// TwinCAT 3 PLC project EOL_TESTER
// ProgramVersion: 3.1.4024.0
// libraries:
//   Tc2_Standard, * (Beckhoff Automation GmbH)
//   Tc2_System, * (Beckhoff Automation GmbH)
//   Tc3_Module, * (Beckhoff Automation GmbH)
// project tree:
//   CustomFBs/Actuator/ FB_ActuatorSimple.TcPOU
//   CustomFBs/Actuator/Structure/ ST_ActuatorConfig.TcDUT, ST_ActuatorInputs.TcDUT, ST_ActuatorOutputs.TcDUT, ST_Actuatorstatus.TcDUT
//   CustomFBs/GateBox/ GateBox_FB.TcPOU, ST_MBMStdInput.TcDUT, ST_MGB2IO.TcDUT
//   CustomFBs/MainSequencer/DUT/ ST_MainSequencerStatus.TcDUT
//   CustomFBs/MainSequencer/ MainSequencer.TcPOU
//   CustomFBs/Motor/ FB_Motor.TcPOU, ST_Motor.TcDUT, ST_MotorInputs.TcDUT, ST_MotorStatus.TcDUT
//   CustomFBs/Rockwell_FB/FileLevel/ COP_Dynamic_String_120.TcPOU, COP_Dynamic_String_15.TcPOU, FLL1_String_120.TcPOU, FLL1_String_15.TcPOU
//   CustomFBs/SequenceStep/ FB_SequenceStep.TcPOU, ST_StepBranch_1.TcDUT
//   CustomFBs/SmartLight_BNI007T/ FB_BNI007T.TcPOU, SmartLight.TcDUT, ST_BNI007T.TcDUT
//   / PlcTask.TcTTO
//   POUs/Cell/ Faulthistory_FB.TcPOU, FB_Cell.TcPOU
//   POUs/Cell/ST_Cell/ ST_Cell.TcDUT, ST_CellFaults.TcDUT, ST_CellMode.TcDUT, ST_Error.TcDUT, ST_Estops.TcDUT, ST_Gates.TcDUT, ST_JobSelection.TcDUT, ST_Power.TcDUT, ST_PV_PB.TcDUT, ST_Safety.TcDUT, ST_SmartLight.TcDUT, ST_Status.TcDUT, ST_Utility.TcDUT
//   POUs/Cell/ST_Station/ ST_StaMode.TcDUT, ST_StaRequest.TcDUT, ST_Stastatus.TcDUT, ST_Station.TcDUT
//   POUs/Effenco/ E_CAN_Effenco.TcDUT
//   POUs/ MAIN.TcPOU
//   POUs/SequenceStep_FB/ SequenceStep_FB.TcPOU, ST_StepBranch.TcDUT
//   POUs/Station/TAP/ E_Checkvalvereject.TcDUT, E_PressureStatus.TcDUT, E_PressureTolerance.TcDUT, E_SenorStatus.TcDUT, E_TapAutoSequenceSteps.TcDUT, FB_TAP.TcPOU
//   POUs/Station/TAP/ST_Tap/ ST_TAP_PB.TcDUT (not stored)
// real-time tasks:
//   TASK PlcTask: cycle T#10ms, priority 20, ADS port 350
// I/O:
//   DEVICE Device 1 (EtherCAT), AmsNetId 5.152.37.14.2.1
//     Term 1 (EK1200) [EK1200-5000 EtherCAT Power supply (2A E-Bus)]
//       Term 2 (EL6070) [EL6070 1Ch. Licensing-Terminal]
//       Term 3 (EL6910) [EL6910, TwinSAFE PLC]
//       Term 4 (EL1918) [EL1918, 8Ch. Safety Input 24V, TwinSAFE]
//         modules: Module 1 (FSOE), Module 2 (FSLOGIC)
//       Term 5 (EL1918) [EL1918, 8Ch. Safety Input 24V, TwinSAFE]
//         modules: Module 1 (FSOE), Module 2 (FSLOGIC)
//       Term 6 (EL2904) [EL2904, 4 Ch. Safety Output 24V, 0.5A, TwinSAFE]
//         modules: Module 1 (FSOES), Module 2 (DO)
//       Term 7 (EL2904) [EL2904, 4 Ch. Safety Output 24V, 0.5A, TwinSAFE]
//         modules: Module 1 (FSOES), Module 2 (DO)
//       Term 8 (EL2904) [EL2904, 4 Ch. Safety Output 24V, 0.5A, TwinSAFE]
//         modules: Module 1 (FSOES), Module 2 (DO)
//       Term 9 (EL2904) [EL2904, 4 Ch. Safety Output 24V, 0.5A, TwinSAFE]
//         modules: Module 1 (FSOES), Module 2 (DO)
//       Term 10 (EL9410) [EL9410 E-Bus Power Supplier  (Diagnostics)]
//       Term 11 (EL1008) [EL1008 8Ch. Dig. Input 24V, 3ms]
//       Term 12 (EL2024) [EL2024 4Ch. Dig. Output 24V, 2A]
//       Term 13 (EL6751) [EL6751 CANopen Master]
//       Term 14 (EL6751) [EL6751 CANopen Master]
//       Term 15 (EL9011) [EL9011 End Terminal]
//   DEVICE Device 2 (EL6751), AmsNetId 5.152.37.14.3.1
//   DEVICE Device 3 (EL6751), AmsNetId 5.152.37.14.4.1

CONFIGURATION EOL_TESTER
    RESOURCE PLC ON TwinCAT3
        TASK PlcTask(INTERVAL := T#10ms, PRIORITY := 20);
        PROGRAM MAIN WITH PlcTask : MAIN;
    END_RESOURCE
END_CONFIGURATION

// ---- CustomFBs/Actuator/Structure/ST_ActuatorConfig.TcDUT
TYPE ST_ActuatorConfig :
STRUCT
	AdvancedFeedbackTimeout		: TON;
	RetractedFeedbackTimeout	: TON := (PT := T#500MS);
	AdvancedDwellTime			: TON;
	RetractedDwellTime			: TON;
END_STRUCT
END_TYPE

// ---- CustomFBs/Actuator/Structure/ST_ActuatorInputs.TcDUT
TYPE ST_ActuatorInputs :
STRUCT
	Advanced  AT%I* : BOOL;
	Retracted AT%I* : BOOL;
END_STRUCT
END_TYPE

// ---- CustomFBs/Actuator/Structure/ST_ActuatorOutputs.TcDUT
TYPE ST_ActuatorOutputs :
STRUCT
	Advance  AT%Q* : BOOL;
	Retract  AT%Q* : BOOL;
END_STRUCT
END_TYPE

// ---- CustomFBs/Actuator/Structure/ST_Actuatorstatus.TcDUT
TYPE ST_Actuatorstatus :
STRUCT
	AdvancedFeedback 	: BOOL;
	RetractedFeedback	: BOOL;
	Advancing			: BOOL;
	Retracting			: BOOL;
END_STRUCT
END_TYPE

// ---- CustomFBs/GateBox/ST_MBMStdInput.TcDUT
TYPE ST_MBMStdInput :
STRUCT
    Run_Mode: BIT;  //
END_STRUCT
END_TYPE

// ---- CustomFBs/GateBox/ST_MGB2IO.TcDUT
TYPE ST_MGB2IO :
STRUCT
    
END_STRUCT
END_TYPE

// ---- CustomFBs/MainSequencer/DUT/ST_MainSequencerStatus.TcDUT
TYPE ST_MainSequencerStatus :
STRUCT
	PowerOn 		: BOOL;
	ResetRequired	: BOOL;
	Auto			: BOOL;
	MaintenanceMode	: BOOL;
END_STRUCT
END_TYPE

// ---- CustomFBs/Motor/ST_Motor.TcDUT
TYPE ST_Motor :
STRUCT
    Start_Safeties              : BOOL; //Start Safety
    Start AT%Q*                 : BOOL; //Start
    Running                     : BOOL; //Running
    Stop                        : BOOL; // Motor Stop
    Manual_Start_PB             : BOOL; //Manual Start PV_PB
    Manual_Stop_PB              : BOOL; //Manual Stop PV_PB
    Start_Fault                 : BOOL; //Start_Fault
    OL_Fault                    : BOOL; //Overload_Fault
    Idle_Standby                : BOOL; //Idle_Standby
    Idle_OFF                    : BOOL; //Idle_OFF
    RunOut                      : BOOL; //RunOut
    ONS                         : R_TRIG; //ONS
    
    Motortimedelay              : TON  := (PT := T#2S); //Motor Timer delay
    MotortimeOFFdelay           : TON;
END_STRUCT
END_TYPE

// ---- CustomFBs/Motor/ST_MotorInputs.TcDUT
TYPE ST_MotorInputs :
STRUCT
    Running  AT %I*  : BOOL;  //Assign with Digital Input EL1008
    Overload AT %I*  : BOOL; 
    Enable   AT %I*  : BOOL;
END_STRUCT
END_TYPE

// ---- CustomFBs/Motor/ST_MotorStatus.TcDUT
TYPE ST_MotorStatus :
STRUCT
    Running : BOOL;
END_STRUCT
END_TYPE

// ---- CustomFBs/SequenceStep/ST_StepBranch_1.TcDUT
TYPE ST_StepBranch_1 :
STRUCT    
    NextStep        : DINT;
    Condition       : ARRAY [1..16] OF BOOL;
    ConditionMet    : BOOL;
END_STRUCT
END_TYPE

// ---- CustomFBs/SmartLight_BNI007T/SmartLight.TcDUT
TYPE SmartLight :
STRUCT
    I: SmartLight_BNI007T;
	O: BYTE;
END_STRUCT
END_TYPE

// ---- CustomFBs/SmartLight_BNI007T/ST_BNI007T.TcDUT
TYPE ST_BNI007T :
STRUCT
  	LC_Ok                   : BOOL; 
	RejectPart              : BOOL;   
	InCycle                 : BOOL;	       
	Req_To_Enter_OK         : BOOL;   
	Req_To_Enter_Requested  : BOOL; 
	All_PP                  : BOOL;       
	No_PP                   : BOOL;
	MaintMode               : BOOL;       
	GateLight               : BOOL;
	OperatorLight           : BOOL;
	Station_Enabled         : BOOL;
	Station_Reset           : BOOL;
	Station_At_Load         : BOOL;
	Ready_For_Unload        : BOOL;
	PP_Not_On_Fault         : BOOL;
	PP_Not_Off_Fault        : BOOL;	
	MachineNotRunning       : BOOL;
	GateLocked              : BOOL;
	GateUnlocked            : BOOL;
	AllGatesReset           : BOOL;  
END_STRUCT
END_TYPE

// ---- POUs/Cell/ST_Cell/ST_Cell.TcDUT
TYPE ST_Cell :
STRUCT
	stMode	        : ST_CellMode;
	stUtility	    : ST_Utility;
	stPower	        : ST_Power;
	Status	        : ST_Status;
	PV_PB	        : ST_PV_PB;
	EStop	        : ST_Estops;
	OperatorLight   : ST_SmartLight;
	Job_Selection   : ST_JobSelection;
    Gates           : ST_Gates;
    Faults          : ST_CellFaults;
    Safety          : ST_Safety;
    
END_STRUCT
END_TYPE

// ---- POUs/Cell/ST_Cell/ST_CellFaults.TcDUT
TYPE ST_CellFaults :
STRUCT
FLT_0:BIT; //***WARNING*** DO NOT USE THIS BIT IN LOGIC!!!
FLT_1:BIT; //SAFETY UNLOCKED IN OMRON SAFETY PLC 
FLT_2:BIT; //ETHERNET COMMUNICATION FAULT
FLT_3:BIT; //ETHERNET SWITCHES - FU#  824 TRIPPED
FLT_4:BIT; 
FLT_5:BIT; //GATE 1 - FU# 832 TRIPPED
FLT_6:BIT; //GATE 2 - FU# 834 TRIPPED
FLT_7:BIT; //STATION MASTER BLOCK - FU# 836 TRIPPED
FLT_8:BIT; //CELL MASTER BLOCK - FU# 839 TRIPPED
FLT_9:BIT; //STA10A VALVE BANK POWER - FU# 902 TRIPPED
FLT_10:BIT; //STA10B VALVE BANK POWER - FU# 904 TRIPPED
FLT_11:BIT; //STA20 VALVE BANK POWER - FU# 912 TRIPPED
FLT_12:BIT; //AIR IS OFF - CHECK MAIN AIR DROP
FLT_13:BIT; //GAS IS OFF - CHECK MAIN GAS SWITCH
FLT_14:BIT; //STATION MB - PORT 0 CONNECTION FAULTED
FLT_15:BIT; //STATION MB - PORT 1 CONNECTION FAULTED
FLT_16:BIT; //STATION MB - PORT 2 CONNECTION FAULTED
FLT_17:BIT; //STATION MB - PORT 3 CONNECTION FAULTED
FLT_18:BIT; //STATION MB - PORT 4 CONNECTION FAULTED
FLT_19:BIT; //STATION MB - PORT 5 CONNECTION FAULTED
FLT_20:BIT; //STATION MB - PORT 6 CONNECTION FAULTED
FLT_21:BIT; //STATION MB - PORT 7 CONNECTION FAULTED
FLT_22:BIT; //CELL MB - PORT 0 CONNECTION FAULTED
FLT_23:BIT; //CELL MB - PORT 1 CONNECTION FAULTED
FLT_24:BIT; //CELL MB - PORT 2 CONNECTION FAULTED
FLT_25:BIT; //CELL MB - PORT 3 CONNECTION FAULTED
FLT_26:BIT; //CELL MB - PORT 4 CONNECTION FAULTED
FLT_27:BIT; //CELL MB - PORT 5 CONNECTION FAULTED
FLT_28:BIT; //CELL MB - PORT 6 CONNECTION FAULTED
FLT_29:BIT; //CELL MB - PORT 7 CONNECTION FAULTED
FLT_30:BIT; 
FLT_31:BIT; 
FLT_32:BIT; 
FLT_33:BIT; 
FLT_34:BIT; 
FLT_35:BIT; 
FLT_36:BIT; 
FLT_37:BIT; 
FLT_38:BIT;
FLT_39:BIT;
FLT_40:BIT; //HMI ESTOP WAS DEPRESSED
FLT_41:BIT; //HMI ESTOP INPUTS INCONSISTENT
FLT_42:BIT; //MHR1 LOCAL ESTOP WAS DEPRESSED
FLT_43:BIT; //MHR1 LOCAL ESTOP INPUTS INCONSISTENT
FLT_44:BIT;
FLT_45:BIT; //OPERATOR ESTOP WAS DEPRESSED
FLT_46:BIT; //OPERATOR ESTOP INPUTS INCONSISTENT
FLT_47:BIT; //OPERATOR 2 RH ESTOP WAS DEPRESSED
FLT_48:BIT; //OPERATOR 2 RH ESTOP INPUTS INCONSISTENT
FLT_49:BIT;
FLT_50:BIT; //GATE 1 ESTOP WAS DEPRESSED
FLT_51:BIT; //GATE 2 ESTOP WAS DEPRESSED
FLT_52:BIT; 
FLT_53:BIT; 
FLT_54:BIT; 
FLT_55:BIT; 
FLT_56:BIT; 
FLT_57:BIT; 
FLT_58:BIT; 
FLT_59:BIT;
FLT_60:BIT; 
FLT_61:BIT; 
FLT_62:BIT; 
FLT_63:BIT; 
FLT_64:BIT;
FLT_65:BIT; 
FLT_66:BIT; 
FLT_67:BIT; 
FLT_68:BIT; 
FLT_69:BIT; //SAFETY GATE 1 NOT IN RUN MODE
FLT_70:BIT; //SAFETY GATE 1 UNLOCKED
FLT_71:BIT; 
FLT_72:BIT; //SAFETY GATE 1 DOOR OPENED
FLT_73:BIT; 
FLT_74:BIT; //SAFETY GATE 2 NOT IN RUN MODE
FLT_75:BIT; //SAFETY GATE 2 UNLOCKED
FLT_76:BIT; 
FLT_77:BIT; //SAFETY GATE 2 DOOR OPENED
FLT_78:BIT; 
FLT_79:BIT; 
FLT_80:BIT; //LIGHT CURTAIN INPUTS INCONSISTENT
FLT_81:BIT; //LIGHT CURTAIN EDM ERROR
FLT_82:BIT; //LIGHT CURTAIN NOT OK
FLT_83:BIT; //LIGHT CURTAIN IN ERROR STATE
FLT_84:BIT; 
FLT_85:BIT; 
FLT_86:BIT; 
FLT_87:BIT; 
FLT_88:BIT; 
FLT_89:BIT; //OMRON SAFETY PROCESSOR NOT MATCHING 
FLT_90:BIT; //HMI POINT IO - COMMUNICATION FAULT
FLT_91:BIT; //OMRON SAFETY PLC - COMMUNICATION FAULT
FLT_92:BIT; //STATION MASTER IO BLOCK - COMMUNICATION FAULT
FLT_93:BIT; //CELL MASTER IO BLOCK - COMMUNICATION FAULT
FLT_94:BIT; //SAFETY GATE 1 - COMMUNICATION FAULT
FLT_95:BIT; //SAFETY GATE 2 - COMMUNICATION FAULT
END_STRUCT
END_TYPE

// ---- POUs/Cell/ST_Cell/ST_CellMode.TcDUT
TYPE ST_CellMode :
STRUCT
	Manual 				: BOOL;         //IN MANUAL MODE
	Auto				: BOOL;         //IN AUTO MODE
	Supervisor_Mode 	: BOOL;         //IN SUPERVISOR MODE
    AutoSelect_Toggle   : um_Toggle;    //Auto Select Toggle
    Autoinitiate         :BOOL;          //Cell Auto Initiate
	In_DryCycle_Select 	: BOOL;         //IN DRY CYCLE MODE
	DryCycle_Runout		: BOOL;         //DRY CYCLE RUN OUT
	DryCycle_ONS		: R_TRIG;       //DRY CYCLE (ONE SHOT)
	In_Continuous_Run	: BOOL;         //IN CONTINUOUS RUN
	Continuos_Run_ONS	: R_TRIG;       //CONTINUOUS RUN (ONE SHOT)
END_STRUCT
END_TYPE

// ---- POUs/Cell/ST_Cell/ST_Error.TcDUT
TYPE ST_Error :
STRUCT
    Active      : BOOL;
    Message     : STRING;
    Priority    : UDINT;
END_STRUCT
END_TYPE

// ---- POUs/Cell/ST_Cell/ST_Estops.TcDUT
TYPE ST_Estops :
STRUCT
Gate1:BIT; 
Gate2:BIT; 
Gate3:BIT; 
Gate4:BIT; 
Gate5:BIT; 
Gate6:BIT; 
Oper1:BIT; 
Oper2:BIT; 
Oper3:BIT; 
Oper4:BIT; 
Oper5:BIT; 
Oper6:BIT; 
Main_Panel:BIT; 
HMI_Panel:BIT; 
Any_EStop_PB_Pressed: BIT;
Local_EStop_1_PB_Pressed: BIT;
END_STRUCT
END_TYPE

// ---- POUs/Cell/ST_Cell/ST_Gates.TcDUT
TYPE ST_Gates :
STRUCT
    //Gate Box
    Request_To_Enter             : BOOL;                  //Request to Enter
    Reset                        : ARRAY [1..5] OF BOOL;  //Reset Door
    Resume_ONS                   : R_TRIG;                //Resume(One Shot)
    OK_To_Enter                  : BOOL;                  //Ok to Enter (Station)
    EntryGranted                 : BOOL;                  //Granted (Unlock Doors)
    EStop_Mem                    : BOOL;
    Closed                       : BOOL;
    Teach_Mode_OK                : BOOL; 
    
    //Gate SAFTY OUTPUT
    DoorUnlockRequest            : ARRAY [1..5] OF BOOL; //Door Unlock Request
    DoorOktoUnlock               : ARRAY [1..5] OF BOOL; //Door Ok to Unlcok
    ReqtoEnterInput_LT  AT%Q*    : ARRAY [1..5] OF BOOL; //WHITE Light  Requst to Enter (Input)     
    FaultResetInput_LT  AT%Q*    : ARRAY [1..5] OF BOOL; //RED Light    Door Fault Reset
    PowerOn_LT          AT%Q*    : ARRAY [1..5] OF BOOL; //GREEN Light  Door Power ON/Cycle start Input
    
    //Gate SAFETY INPUT
    Run_Mode                                    : BIT;//SI_RM
	Connection_Fauled                           : BIT;//SI_CF
	Diagnostic_Active                           : BIT;//SI_DA
	FailSafe_Input_EStop_OK                     : BIT;//SI_FIES
	FailSafe_Input_DoorPosition                 : BIT;//SI_FI_D
	FailSafe_Input_BoltPosition                 : BIT;//SI_FI_B
	FailSafe_Input_GuardLocking                 : BIT;//SI_FI_L (GATE LOCKED)
	FailSafe_Input_DoorAndBolt_Position         : BIT;//SI_FI_SK
	FailSafe_Input_DoorBoltAndGuardLocking      : BIT;//SI_FI_UK
	Maintenance_Mode                            : BIT;//SI_S94
    DoorReqtoEnterInput AT%I*                   : ARRAY [1..5] OF BOOL; //SI_S2//WHITE PB  Requst to Enter (Input)     
    DoorFaultResetInput AT%I*                   : ARRAY [1..5] OF BOOL; //SI_S3//RED PB    Door Fault Reset
    DoorPowerOn         AT%I*                   : ARRAY [1..5] OF BOOL; //SI_S4//GREEN PB  Door Power ON/Cycle start Input
	Diagnostics_Plausibility_Fault              : BIT;//SI_D_PF
	Diagnostics_Emergency_Stop                  : BIT;//SI_D_ES
	Diagnostics_GuardLocking                    : BIT;//SI_D_OL
	Diagnostics_Lifetime                        : BIT;//SI_D_LT

    
END_STRUCT                          
END_TYPE

// ---- POUs/Cell/ST_Cell/ST_JobSelection.TcDUT
TYPE ST_JobSelection :
STRUCT
Auto_Job_Mode			: BOOL;
Part_Sel_Chng_OK		: BOOL;
HMI_Selected_Job		: DINT;
Job_Number_Selected		: DINT;
Job_Number_Selected_Last: DINT;
Job_Change_Started		: BOOL;
Job_Change_Delay		: TON;	
END_STRUCT
END_TYPE

// ---- POUs/Cell/ST_Cell/ST_Power.TcDUT
TYPE ST_Power :
STRUCT
Gen_Safety	:BOOL;		//General_Safety_OK(COntrol POwer)(Gate Closed)(Air OK)
PowerOn		:BOOL; 		//CONTROL POWER ON
EStops		:ST_Estops;	//NO E-STOPS BUTTONS PRESSED
GatesClosed	:BOOL; 		//CELL SAFETY GATES CLOSED & RESET
END_STRUCT
END_TYPE

// ---- POUs/Cell/ST_Cell/ST_PV_PB.TcDUT
TYPE ST_PV_PB :
STRUCT
	FaultReset_PB 		:BOOL;  //FAULT_RESET PV_PB
	AutoManual_SS 		:BOOL; 	//AUTO/MANUAL SELECTOR SWITCH PV PB
	AutoSelector_PB 	:BOOL; 	//AUTO_SELECTOR SWITCH PV PB
	ManualSelector_PB 	:BOOL; 	//MANUAL_SELECTOR SWITCH PV PB
	AutoMode_PB		:BOOL; 	//AUTO MODE PV PB
	Dry_Cycle_Mode		:BOOL;	//DRY_CYCLE_MODE PV PB
	ContinousRun_Mode	:BOOL;	//CONTINUOUS RUN MODE PV PB
	FaultHistory_Reset	:BOOL;	//FAULT HISTOTY RESET PV PB
END_STRUCT
END_TYPE

// ---- POUs/Cell/ST_Cell/ST_Safety.TcDUT
TYPE ST_Safety :
STRUCT
    MCPEstopOk AT%I*  : BOOL;
    SafetyOk AT%I*    : BOOL;
    
END_STRUCT
END_TYPE

// ---- POUs/Cell/ST_Cell/ST_SmartLight.TcDUT
TYPE ST_SmartLight :
STRUCT
	Green			: BOOL;  
	Process_Fault	: BOOL;
	InCycle			: BOOL;
	Blue			: BOOL;
	Orange			: BOOL;
	White			: BOOL;
    Flash			: BOOL;	
END_STRUCT
END_TYPE

// ---- POUs/Cell/ST_Cell/ST_Status.TcDUT
TYPE ST_Status :
STRUCT
AllComms_OK		:BOOL; //ALL COMMUNICATION MODULES OK
ENetComms_OK    :BOOL; //All EtherCAT Comms Ok
Faulted			:BOOL; //Fault(s) Present
Fault_Reset		:BOOL; //Fault Reset
All_Faults		:BOOL; //ANY STATION FAULTED
All_in_Auto		:BOOL; //ALL_STATIONS IN AUTO MODE
All_in_Manuals	:BOOL; //ALL_SATIONS_IN MANUAL MODE
StationsHeld	:BOOL; //Station is Hold in between Test
Held			:BOOL; //CELL HOLD BUTTON PRESSED
Message			:BOOL; //Message(s) Present
ProcessOn		:BOOL; //DUT (Device Under Test) is ON
ProcessOff		:BOOL; //DUT (Device Under Test) is OFF
OKToEnterGates	:BOOL; //Safe
END_STRUCT
END_TYPE

// ---- POUs/Cell/ST_Cell/ST_Utility.TcDUT
TYPE ST_Utility :
STRUCT
MainAirOn	     :BOOL;        //MAIN AIR PRESSURE OK
MainAirPSI AT%I* :REAL;        //MAIN AIR DATA FROM BALLUFF PRESSURE SENSOR
END_STRUCT
END_TYPE

// ---- POUs/Cell/ST_Station/ST_StaMode.TcDUT
TYPE ST_StaMode :
STRUCT
    ManualReady             : BIT; //READY FOR MANUAL
    Manual                  : BIT;//IN MANUAL MODE
    AutoReady               : BIT; //READY FOR AUTO
    Auto                    : BIT; //IN AUTO MODE
    DryCycleReady           : BIT; // READY FOR DRYCYCLE
    DryCycle                : BIT; //IN DRY CYCLE MODE (RUN EMPTY)
    PartTest                : BIT; //WHITE RABBIT TEST MODE
    AutoWarning             : TON; // AUTO WARNING TIMER
    Job_Select_PB           : BIT;// JOB SELECT PUSHBUTTON
END_STRUCT
END_TYPE

// ---- POUs/Cell/ST_Station/ST_StaRequest.TcDUT
TYPE ST_StaRequest :
STRUCT
    AutoInitiate        : BIT; // 
    AutoConfirm         : BIT; // 
    FaultReset          : BIT; // 
    Hold                : BIT; // 
    LampTest            : BIT; // 
    PauseMSG            : BIT; // 
    DryCycle            : BIT; // 
    AllProcessOn        : BIT; // 
    AllProcessOff       : BIT; // 
    ProdCountReset      : BIT; //   
END_STRUCT
END_TYPE

// ---- POUs/Cell/ST_Station/ST_Stastatus.TcDUT
TYPE ST_Stastatus :
STRUCT
    AirOff                  : BIT; // 
    AirOn                   : BIT; // 
    AllParts                : BIT; // STATION HAS ALL PARTS PRESENT 
    AllProcessesComplete    : BIT; // ALL PROCESSES COMPLETE
    All_Tools_In_Known_Pos  : BIT; //
    All_Faults              : BIT;// 
    Auto                    : BIT; // STATION IN AUTO
    ClearForTransfer        : BIT; // 
    CommOK                  : BIT; // STATION COMMUNICATIONS ARE OK
    DryCycle                : BIT; // STATION IN DRY CYCLE
    Faulted                 : BIT; // STATION FAULTED
    GasFlowOff              : BIT; // 
    GasFlowOn               : BIT; // 
    Held                    : BIT; // STATION HELD
    HoldActive              : BIT; // STATION HOLD IS ACTIVE
    Home                    : BIT; // TOOL AT HOME POSITION
    InCycle                 : BIT; // STATION IN CYCLE
    Load1                   : BIT; // TOOL AT LOAD POSITION 1
    Load2                   : BIT; // TOOL AT LOAD POSITION 2
    Manual                  : BIT; // STATION IN MANUAL
    Message                 : BIT; // Message(s) Present
    NoParts                 : BIT; // STATION HAS NO PARTS PRESENT
    NoProcComp              : BIT; // NO PROCESS COMPLETE
    NotClear                : BIT; // 
    OK_To_Enter             : BIT; // Clear To Enter if Gate Request Has Been Made
    PartPres                : BIT; // 
    Proc1Comp               : BIT; // 1st PROCESS COMPLETE
    Proc2Comp               : BIT; // 2nd PROCESS COMPLETE
    Proc3Comp               : BIT; // 3rd PROCESS COMPLETE
    Proc4Comp               : BIT; // 4th PROCESS COMPLETE
    Proc5Comp               : BIT; // 5th PROCESS COMPLETE
    Proc6Comp               : BIT; // 6th PROCESS COMPLETE
    Proc7Comp               : BIT; // 7th PROCESS COMPLETE
    Proc8Comp               : BIT; // 8th PROCESS COMPLETE
    ProcEnbld               : BIT; // 
    ProcNotEnbld            : BIT; // 
    Sla01_ID                : BYTE; // ID PRESENT ON SLAVE#1
    Sla02_ID                : BYTE; // ID PRESENT ON SLAVE#2
    SteppersReset           : BIT; // 
    Tool_Monitor            : DINT;
    Unload1                 : BIT; // TOOL AT UNLOAD POSITION 1
    UnLoad2                 : BIT; // TOOL AT UNLOAD POSITION 2
    WaterFlowOff            : BIT; // 
    WaterFlowOn             : BIT; // 
    Work1                   : BIT; // TOOL AT WORK POSITION 1
    Work2                   : BIT; // TOOL AT WORK POSITION 2
    Work3                   : BIT; // TOOL AT WORK POSITION 3
END_STRUCT
END_TYPE

// ---- POUs/Cell/ST_Station/ST_Station.TcDUT
TYPE ST_Station :
STRUCT
    Mode        : ST_StaMode;                   // Station Mode
    Status      : ST_Stastatus;                // Station Status 
    Req         : ST_StaRequest;               // 
END_STRUCT
END_TYPE

// ---- POUs/Effenco/E_CAN_Effenco.TcDUT
{attribute 'qualified_only'}
{attribute 'strict'}
TYPE E_CAN_Effenco :
(
	enum_member := 0
);
END_TYPE

// ---- POUs/SequenceStep_FB/ST_StepBranch.TcDUT
TYPE ST_StepBranch :
STRUCT    
    NextStep        : DINT;
    Condition       : ARRAY [1..16] OF BOOL;
    ConditionMet    : BOOL;
END_STRUCT
END_TYPE

// ---- POUs/Station/TAP/E_Checkvalvereject.TcDUT
{attribute 'qualified_only'}
{attribute 'strict'}
TYPE E_Checkvalvereject :
(
	enum_member         := 0,
    CheckvalveOk        := 10,
    Checkvalvefailure   := 20
);
END_TYPE

// ---- POUs/Station/TAP/E_PressureStatus.TcDUT
{attribute 'qualified_only'}
{attribute 'to_string'}
TYPE E_PressureStatus : 
(
    FillingupTestFail    := 10,
    FillingupTestPass    := 20,
    PressuretestOk       := 30,
    Pressuretestfail     := 40,
    InletLeakDetect      := 50,
    OilLeakDetect        := 60
    	
);
END_TYPE

// ---- POUs/Station/TAP/E_PressureTolerance.TcDUT
{attribute 'qualified_only'}
{attribute 'strict'}
TYPE E_PressureTolerance :
(
	enum_member := 0
);
END_TYPE

// ---- POUs/Station/TAP/E_SenorStatus.TcDUT
{attribute 'qualified_only'}
{attribute 'strict'}
TYPE E_SenorStatus :
(
	enum_member         := 0,
    P1UUTSensorOK       := 10,
    P1UUTSensorFail     := 20,
    P2UUTSensorOK       := 30,
    P2UUTSensorFail     := 40,
    Filterisdetected    := 50,
    Filterismissing     := 60
    
    
);
END_TYPE

// ---- POUs/Station/TAP/E_TapAutoSequenceSteps.TcDUT
{attribute 'qualified_only'}
{attribute 'strict'}
TYPE E_TapAutoSequenceSteps :
(
	STARTING_CONDITIONS		    := 10,
    START_FILLING_PHASE 	    := 20,
	TE_RUN_MOTOR			    := 30,
//	TE_MOTOR_START_DELAY	    := 40,
	START_UUT_MOTOR			    := 50,
	UUT_MOTOR_DELAY			    := 60,
	INITIAL_PRESSURE_TEST	    := 70,
    TE_STOP_MOTOR               := 80,
    STOP_UUT_MOTOR              := 90,
    END_FILLING_PHASE           := 100,
    START_STATIC_PRESSURE_TEST  := 110,
    OUTLET_PRESSURE_TEST        := 120,
    OIL_LEAK_TEST               := 130,
    END_STAITC_PRESSURE_TEST    := 140,
    START_FUNCTIONAL_TEST       := 150,
    UUT_SENSOR_CHECK            := 160,
    END_FUNCTIONAL_TEST         := 170,
    START_TAP_CHECKVALVE_TEST   := 180,
    CHECK_VALVE_TEST            := 190,
    END_TAP_CHECKVALVE_TEST     := 200,
    START_DRAINING_TEST         := 210, 
    STOP_DRAINING_TEST          := 220,    
    COMPLETE                := 1000
	
);
END_TYPE

// ---- POUs/MAIN.TcPOU
PROGRAM MAIN
VAR
END_VAR

END_PROGRAM

// ---- CustomFBs/Actuator/FB_ActuatorSimple.TcPOU
FUNCTION_BLOCK FB_ActuatorSimple
VAR_INPUT
    stCell      : ST_Cell;
    stStation   : ST_Station;
END_VAR
VAR
	stStatus			: ST_Actuatorstatus;
	stConfiguration 	: ST_ActuatorConfig;
	stInputs			: ST_ActuatorInputs;
	stOutputs			: ST_ActuatorOutputs;
END_VAR

//_M_EvaluateInputs();
_M_Status();

METHOD PRIVATE _M_EvaluateInputs
VAR_INPUT
END_VAR
END_METHOD

METHOD PUBLIC _M_Status : BOOL
VAR_INPUT
END_VAR
// Reset Status
//Status.AdvancedFeedback := FALSE;
//Status.Advancing := FALSE;
//Status.RetractedFeedback := FALSE;
//Status.Retracting := FALSE;

// Set According To Raw Value
IF stInputs.Advanced AND NOT stInputs.Retracted THEN
    stStatus.AdvancedFeedback := TRUE;
    stConfiguration.AdvancedFeedbackTimeout(IN:=FALSE);
    IF stOutputs.Advance THEN
        stOutputs.Advance := FALSE;
    END_IF
ELSE
    IF stOutputs.Advance THEN
        stStatus.Advancing := TRUE;
    END_IF
END_IF	

IF stInputs.Retracted AND stInputs.Advanced THEN 	
    stStatus.RetractedFeedback := TRUE;
    IF stOutputs.Retract THEN
        stOutputs.Retract := FALSE;
    END_IF
ELSE
    IF stOutputs.Retract THEN
        stStatus.Retracting := TRUE;
    END_IF
END_IF

IF stInputs.Advanced AND stInputs.Retracted THEN
    //error handling
END_IF
END_METHOD

METHOD PUBLIC M_Advance
//At Advance Position

IF stStatus.RetractedFeedback AND NOT stStatus.AdvancedFeedback THEN      
      stOutputs.Retract := FALSE;
      stOutputs.Advance := TRUE;
      stConfiguration.AdvancedFeedbackTimeout(IN:=TRUE);
END_IF      
IF NOT stStatus.AdvancedFeedback AND stConfiguration.AdvancedFeedbackTimeout.Q THEN
    //time out happened - indicate fault
    //reset output for advance and retract
    //monitor safety
END_IF
END_METHOD

METHOD PUBLIC M_Retract
VAR_INPUT
END_VAR
//At Retract Position
END_METHOD

PROPERTY PUBLIC P_Config : REFERENCE TO ST_ActuatorConfig
GET // PUBLIC
P_Config REF= stConfiguration;
END_GET
END_PROPERTY

PROPERTY PUBLIC P_Status : REFERENCE TO ST_Actuatorstatus
GET
P_Status REF= stStatus;
END_GET
END_PROPERTY

END_FUNCTION_BLOCK

// ---- CustomFBs/GateBox/GateBox_FB.TcPOU
FUNCTION_BLOCK GateBox_FB
VAR 
    Gate1   : ST_Gates;
    Gate2   : ST_Gates;
END_VAR

//GateBox-1 Lock Solenoid
IF GVL.stCell.Gates.DoorReqtoEnterInput[1] AND GVL.stCell.Gates.Request_To_Enter THEN
    GVL.stCell.Gates.DoorUnlockRequest[1] := TRUE;
ELSIF GVL.stCell.Gates.DoorPowerOn[1] AND  GVL.zz_Deep.0 AND GVL.zz_Deep.0 THEN
    GVL.stCell.Gates.DoorUnlockRequest[1] := FALSE;
END_IF

GVL.stCell.Gates.DoorOktoUnlock[1] := (GVL.stCell.Gates.EntryGranted OR 
                                          GVL.stCell.Gates.DoorOktoUnlock[1] OR 
                                          GVL.zz_Deep.0)  AND 
                                          GVL.stCell.Gates.DoorUnlockRequest[1];
                                         
//GateBox-1 - Smart light Mapping
//White Light
GVL.stCell.Gates.ReqtoEnterInput_LT[1] :=  GVL.stCell.Gates.DoorUnlockRequest[1] AND 
                                            GVL.stCell.Gates.Request_To_Enter AND 
                                            GVL.stCell.Gates.OK_To_Enter AND 
                                            GVL.stCell.Gates.EntryGranted AND 
                                            (NOT Gate1.Maintenance_Mode OR (Gate1.Maintenance_Mode AND Gate1.Teach_Mode_OK));  

//Green Liight
GVL.stCell.Gates.FaultResetInput_LT[1] :=  (Gate1.Reset OR (Gate1.closed AND NOT Gate1.Reset AND Gate1.Maintenance_Mode) AND 
                                            (NOT Gate1.Maintenance_Mode OR (Gate1.Maintenance_Mode AND Gate1.Teach_Mode_OK)))  OR
                                            (Gate1.Maintenance_Mode AND NOT Gate1.Teach_Mode_OK);
                                            
                                            
//Red Light
GVL.stCell.Gates.FaultResetInput_LT[1] :=  (GVL.stCell.Status.All_Faults AND 
                                            ( NOT Gate1.Maintenance_Mode OR (Gate1.Maintenance_Mode AND Gate1.Teach_Mode_OK))) OR
                                            Gate1.DoorFaultResetInput   OR
                                            (Gate1.Maintenance_Mode AND NOT Gate1.Teach_Mode_OK);
                                            

                                            
                                            
                                            
                                            
//GateBox-2 Lock Solenoid
IF GVL.stCell.Gates.DoorReqtoEnterInput[2] AND GVL.stCell.Gates.Request_To_Enter THEN
    GVL.stCell.Gates.DoorUnlockRequest[2] := TRUE;
ELSIF GVL.stCell.Gates.DoorPowerOn[1] AND  GVL.zz_Deep.0 AND GVL.zz_Deep.0 THEN
    GVL.stCell.Gates.DoorUnlockRequest[2] := FALSE;
END_IF

GVL.stCell.Gates.DoorOktoUnlock[2] := (GVL.stCell.Gates.EntryGranted OR 
                                          GVL.stCell.Gates.DoorOktoUnlock[2] OR 
                                          GVL.zz_Deep.0)  AND 
                                          GVL.stCell.Gates.DoorUnlockRequest[2];

//GateBox-2 - Smart light Mapping
//White Light
GVL.stCell.Gates.ReqtoEnterInput_LT[2] :=  GVL.stCell.Gates.DoorUnlockRequest[2] AND 
                                            GVL.stCell.Gates.Request_To_Enter AND 
                                            GVL.stCell.Gates.OK_To_Enter AND 
                                            GVL.stCell.Gates.EntryGranted AND 
                                            (NOT Gate2.Maintenance_Mode OR (Gate2.Maintenance_Mode AND Gate2.Teach_Mode_OK));  

//Green Liight
GVL.stCell.Gates.FaultResetInput_LT[2] :=  (Gate2.Reset OR (Gate2.closed AND NOT Gate2.Reset AND Gate2.Maintenance_Mode) AND 
                                            (NOT Gate2.Maintenance_Mode OR (Gate2.Maintenance_Mode AND Gate2.Teach_Mode_OK)))  OR
                                            (Gate2.Maintenance_Mode AND NOT Gate2.Teach_Mode_OK);
                                            
                                            
//Red Light
GVL.stCell.Gates.FaultResetInput_LT[2] :=  (GVL.stCell.Status.All_Faults AND 
                                            ( NOT Gate2.Maintenance_Mode OR (Gate2.Maintenance_Mode AND Gate2.Teach_Mode_OK))) OR
                                            Gate2.DoorFaultResetInput   OR
                                            (Gate2.Maintenance_Mode AND NOT Gate2.Teach_Mode_OK)

END_FUNCTION_BLOCK

// ---- CustomFBs/MainSequencer/MainSequencer.TcPOU
FUNCTION_BLOCK MainSequencer
VAR_INPUT
	Status	: REFERENCE TO ST_MainSequencerStatus;
END_VAR
VAR
	fbTest1Sequencer	: Test1Sequencer;	
	oPowerPackChargeRequest	 AT%Q* : BOOL;
END_VAR

_M_Test1();
//_M_AutoSequence();

METHOD PRIVATE _M_AutoSequence
VAR_INPUT
END_VAR
fbTest1Sequencer.M_AutoSequence(AutoSteps := E_Test1AutoSteps.PRESSURIZEHYDRAULICMOTOR);
END_METHOD

METHOD PRIVATE _M_Test1
VAR_INPUT
END_VAR
fbTest1Sequencer();
END_METHOD

END_FUNCTION_BLOCK

// ---- CustomFBs/Motor/FB_Motor.TcPOU
FUNCTION_BLOCK FB_Motor
VAR_INPUT
   SafetyOk               : BOOL;
END_VAR
VAR 
    stMotor               : ST_Motor;
    stMotorInputs         : ST_MotorInputs;
    Error                 : ST_Error (Priority := 999);
    Status                : ST_MotorStatus;
END_VAR


(* Monitoring all Digital Inputs during Process *)
M_Monitor();

(* HPU - Faults *)
M_Fault();

METHOD PRIVATE M_Fault : BOOL
VAR_INST
    (*Fault Timers*)
    System_Faults       : ARRAY [0..10] OF BOOL;
	Fault_Tmrs          : ARRAY [0..10] OF TON;
END_VAR
VAR
    Error : ST_Error;
END_VAR
 Error.Active := stMotorInputs.Overload;
 Error.Message := 'Motor Overload Tripped';
 M_RaiseError(InputError := Error);



   (*Fault1 - HPU Enable input not coming on: check relay in MCP Panel*)
		Fault_Tmrs[1].PT:= T#2.5S;
		Fault_Tmrs[1]();
		Fault_Tmrs[1].IN:=  GVL.zz_Deep.0 AND //need to add safety EDM condition 
							  stMotorInputs.Enable ;
        System_Faults[1]:= Fault_Tmrs[1].Q;
        
    (*Fault2 - HPU Running Input is not coming ON *)
		Fault_Tmrs[2].PT:= T#2.5S;
		Fault_Tmrs[2]();
		Fault_Tmrs[2].IN:= stMotor.Start AND
                              stMotorInputs.Running; 
        System_Faults[2]:= Fault_Tmrs[2].Q;    
        
    (*Fault3 - HPU Motor OverLoad Trip: CheckUnit *)
		Fault_Tmrs[3].PT:= T#0.5S;
		Fault_Tmrs[3]();
		Fault_Tmrs[3].IN:= stMotorInputs.Overload;  
        System_Faults[3]:= Fault_Tmrs[].Q;  
        
   (*Fault4 - Low Critical Oil: Motor can not run until Tank is Filled *)
		Fault_Tmrs[].PT:= T#0.5S;
		Fault_Tmrs[]();
		Fault_Tmrs[].IN:= ;  
        System_Faults[]:= Fault_Tmrs[].Q;
        
   (*Fault5 - Oil Temperature Critical: Motor Can not run until Oil Cools Down *)
		Fault_Tmrs[].PT:= T#0.5S;
		Fault_Tmrs[]();
		Fault_Tmrs[].IN:=   
        System_Faults[]:= Fault_Tmrs[].Q;
        
    (*Fault6 - HPU High Pressure Bypass Valve Faulted - not going to Low Pressure: Major Fault *)
		Fault_Tmrs[].PT:= T#12.5S;
		Fault_Tmrs[]();
		Fault_Tmrs[].IN:=  
        System_Faults[]:= Fault_Tmrs[].Q;
END_METHOD

METHOD PRIVATE M_Monitor : BOOL
VAR   
END_VAR

//Do we still need to monitor even if we are monitoring in faults

//IF stMotor.Start  THEN    //Should I add more condition from safety related to CH-1 and CH-2
//     stMotorInputs.Running AND stMotorInputs.Enable AND NOT stMotorInputs.Overoload
  
//END_IF


//Do we need to monitro safety input here as well?
END_METHOD

METHOD PRIVATE M_RaiseError
VAR_INPUT
    InputError : ST_Error;
END_VAR
IF InputError.Priority < Error.Priority THEN
    Error := InputError;
END_IF
END_METHOD

METHOD PUBLIC M_ResetFault
VAR
    NullError : ST_Error;
END_VAR
Error := NullError;
END_METHOD

METHOD M_Start : BOOL
VAR

    SafetyNOKError : ST_Error (Message := 'Motor Not Started Fault Due To Safety NOK', Priority := 1); 
    
END_VAR
 //Verify Motor Safety
 
(*IF  SafetyOk  AND                                 //tHIS CONDITION WILL MONITOR BEFORE RUN MOTOR PROGRAM    
         NOT stMotorInputs.Overload AND            //OL Relay Tripped Input
         NOT M_Fault(); THEN                    //Need to verify this logic
    stMotor.Start_Safeties := TRUE;
ELSE
    stMotor.Start_Safeties := FALSE;
END_IF*)          
         
IF (stStation.Mode.Auto OR    
         (stStation.Mode.Manual AND 
            stMotor.Manual_Start_PB)) AND 
                stMotor.Start_Safeties THEN
    stMotor.Start := TRUE;
    stmotor.Motortimedelay (IN := TRUE);   
ELSE
     

IF SafetyOk THEN
    stMotor.Start := TRUE;
ELSE    
    stMotor.Start := FALSE;
    SafetyNOKError.Active := TRUE;
    M_RaiseError(InputError := SafetyNOKError);
END_IF
END_METHOD

METHOD M_Stop : BOOL
VAR_INST
    
END_VAR
 //Verify Motor Safety
 
IF  fbCell.M_Power() AND fbCell.M_Utility() AND 
         GVL.zz_Deep  AND                          //safety needs to add    
         NOT stHPU_Input AND                      //OL Relay Tripped Input
         NOT M_Fault(); THEN                      //Need to verify this logic
    stMotor.Start_Safeties := TRUE;
ELSE
    stMotor.Start_Safeties := FALSE;
END_IF         
         
IF (stStation.Mode.Auto OR    
         (stStation.Mode.Manual AND 
            stMotor.Manual_Stop_PB)) AND 
                stMotor.Start_Safeties THEN
    stMotor.Stop := TRUE;
    stMotor.MotortimeOFFdelay (IN := TRUE);   
ELSE

IF stMotor.Stop AND stmotor.MotortimeOFFdelay.Q AND NOT stMotor.Motortimedelay.Q   THEN
     //time out happended - indicate fault
     //reset outout for coil
     //monitor safety
END_IF
END_IF
END_METHOD

PROPERTY P_Status : ST_MotorStatus
GET
P_Status := Status;
END_GET
END_PROPERTY

END_FUNCTION_BLOCK

// ---- CustomFBs/Rockwell_FB/FileLevel/COP_Dynamic_String_120.TcPOU
FUNCTION_BLOCK COP_Dynamic_String_120
VAR_IN_OUT
	Source: ARRAY[*] OF STRING(120);
	Dest: ARRAY[*] OF STRING(120);
END_VAR
VAR_INPUT
	SStart: DINT;
	DStart: DINT;
	Length: BYTE;
END_VAR
VAR_OUTPUT
END_VAR
VAR
	i: BYTE;
END_VAR

FOR i := 0 TO Length DO
	Dest[i+DStart]:= Source[i+SStart];
END_FOR

END_FUNCTION_BLOCK

// ---- CustomFBs/Rockwell_FB/FileLevel/COP_Dynamic_String_15.TcPOU
FUNCTION_BLOCK COP_Dynamic_String_15
VAR_IN_OUT
	Source: ARRAY[*] OF STRING(15);
	Dest: ARRAY[*] OF STRING(15);
END_VAR
VAR_INPUT
	SStart: DINT;
	DStart: DINT;
	Length: BYTE;
END_VAR
VAR_OUTPUT
END_VAR
VAR
	i: BYTE;
END_VAR

FOR i := 0 TO Length DO
	Dest[i+DStart]:= Source[i+SStart];
END_FOR

END_FUNCTION_BLOCK

// ---- CustomFBs/Rockwell_FB/FileLevel/FLL1_String_120.TcPOU
FUNCTION_BLOCK FLL1_String_120
VAR_IN_OUT
	Dest: ARRAY[*] OF STRING(120);
END_VAR
VAR_INPUT
	Source: STRING;
	Start: DINT;
	Length: DINT;
END_VAR
VAR_OUTPUT
END_VAR
VAR
	i: DINT;	
END_VAR

FOR i:= 0 TO Length DO
	Dest[i + Start]:= Source;
END_FOR

END_FUNCTION_BLOCK

// ---- CustomFBs/Rockwell_FB/FileLevel/FLL1_String_15.TcPOU
FUNCTION_BLOCK FLL1_String_15
VAR_IN_OUT
	Dest: ARRAY[*] OF STRING(15);
END_VAR
VAR_INPUT
	Source: STRING;
	Start: DINT;
	Length: DINT;
END_VAR
VAR_OUTPUT
END_VAR
VAR
	i: DINT;	
END_VAR

FOR i:= 0 TO Length DO
	Dest[i + Start]:= Source;
END_FOR

END_FUNCTION_BLOCK

// ---- CustomFBs/SequenceStep/FB_SequenceStep.TcPOU
FUNCTION_BLOCK FB_SequenceStep
VAR_INPUT
    Branch          : ARRAY [1..16] OF ST_StepBranch;
END_VAR
VAR_OUTPUT    
    CurrentStep     : DINT;    
    Entry           : BOOL := TRUE;
END_VAR
VAR
    i : SINT;
    j : SINT;
    Firstscan : BOOL := TRUE;
END_VAR

Entry := FALSE;

IF FirstScan THEN
    Initialize:
    FOR i:= 1 TO 16 DO
        FOR j:= 1 TO 16 DO
            Branch[i].Condition[j] := TRUE;
        END_FOR    
	END_FOR
    Firstscan := FALSE; 
    RETURN;   
END_IF

FOR i:= 1 TO 16 DO
    Branch[i].ConditionMet := TRUE;
    FOR j:= 1 TO 16 DO        
        Branch[i].ConditionMet := Branch[i].Condition[j] AND Branch[i].ConditionMet;
	END_FOR
    IF Branch[i].ConditionMet THEN        
        CurrentStep := Branch[i].NextStep;
        Entry := TRUE;
        JMP Initialize;
	END_IF
    //
END_FOR

END_FUNCTION_BLOCK

// ---- CustomFBs/SmartLight_BNI007T/FB_BNI007T.TcPOU
FUNCTION_BLOCK FB_BNI007T
VAR_INPUT
    stLightData         : ST_BNI007T;
    ECAT_MB_Address     : UINT;	
    MB_Port_Num         : UINT;  // Port1=0 ... Port8=7
END_VAR
VAR_OUTPUT
    Mapped_SmartLight   : BYTE;  //001 = Green, 010 = Process_Fault, 011 = InCycle, 100 = Blue, 101 = Orange, 110= Purple/User Defined (254,0,254), 111= White
END_VAR
VAR
    GateLightMode       : BOOL;
	OpLightMode         : BOOL;
	Flash               : BOOL;	        
	Green               : BOOL;
	Red                 : BOOL;
	Yellow              : BOOL;
	Blue                : BOOL;
	Orange              : BOOL;
	Purple              : BOOL;
	White               : BOOL;
	All_PP_OK           : BOOL;
	PartMissing         : BOOL;
	OpClearToEnter      : BOOL;
	PartNotRemoved      : BOOL;
	MachineActive       : BOOL;
	MachineInActive     : BOOL;
	RejectPart          : BOOL;
	RTE_Req             : BOOL;
	RTE_OK              : BOOL;
	MaintModeActive     : BOOL;
	Gates_OK            : BOOL;
	GateOpen            : BOOL;
	Runlight_Mode       : BOOL;
	Segment_Mode        : BOOL;
	//Mode_Select_Message : IOL_Azylic_Communication_v11;
	StartModeMsg        : BOOL;
	ResetMsg            : BOOL;	// 
	Write_Mode          : BOOL;
	MsgExecInProgress   : BOOL;
	MsgExecError        : BOOL;
	MsgExecErrCode      : UINT;
	ReadData            : ARRAY [0..231] OF BYTE;
	WriteData           : ARRAY [0..19] OF BYTE;
	ReadTmr             : ARRAY[0..5] OF TON;
	ReadET              : ARRAY[0..5] OF TIME;
	ONS                 : ARRAY[0..31] OF R_TRIG;
	MsgExecDN           : BOOL;
	debug               : DINT;
	Index               : UINT;
	Enable_Read         : BOOL;
	Reset_Write_Tmr     : TON;
	Reset_Read_Tmr      : TON;
	Reset_Start_Mode_Select_Tmr: TON;
	// True = Write Data, False = Read Data
	Enable_Write_Mode   : BOOL;
	Read_Mode           : BOOL;
	Wait_For_Read       : BOOL;
	Enable_Write        : BOOL;
	Prev_Color          : BYTE;
	StopWriteCmd        : BOOL;
	StopRunLightModeCmd : BOOL;
	StopSegmentModeCmd  : BOOL;
	Write_Color         : BOOL;
	ModeSelectMsgCycle  : um_Cycle;
	CycleTON            : ARRAY[0..9] OF TON;
	CycleTOF            : ARRAY[0..9] OF TOF;
	StartedModeMsg      : BOOL;
	ModeMsgExecuted     : BOOL;
	Enable_Read_Mode    : BOOL;
	ColorSelectMsgCycle : um_Cycle;
	ColorMsgExecuted    : BOOL;
	TON_0               : TON;
	//Bit_Distribute_FB   : COP_Dynamic_BYTE;
	Color               : BYTE;
	ReadColor           : BYTE;
	StartColorMsg       : BOOL;
	StartedColorMsg     : BOOL;
	StartMsg            : BOOL;
END_VAR

//Mode Selsection
(*
IF LightData.OperatorLight THEN
    OpLightMode :=TRUE;
END_IF

GateLightMode  := LightData.GateLight;
All_PP_OK      := LightData.Station_Enabled AND LightData.Station_Reset AND LightData.All_PP;
PartMissing    := LightData.Station_Enabled AND LightData.Station_Reset AND NOT LightData.All_PP AND LightData.No_PP;
OpClearToEnter := LightData.Station_At_Load AND LightData.Station_Enabled AND (LightData.Station_Reset OR LightData.Ready_For_Unload);
RejectPart     := LightData.Station_Enabled AND LightData.RejectPart;
MachineInActive:= LightData.MachineNotRunning;

//Mapping to Light Color for Operator
White          := All_PP_OK OR PartMissing;
Red            := RejectPart;
Green          := OpClearToEnter;
Blue           := MachineActive;
Yellow         := MachineActive;
Flash          := PartMissing OR RejectPart OR PartNotRemoved;

//Mapping to Light Color For Gates
//Gate Lights
//Condition for Gate Open
GateOpen := NOT LightData.MaintMode AND LightData.GateUnlocked;
RTE_Req  := LightData.Req_To_Enter_Requested AND LightData.GateLocked AND NOT LightData.Req_To_Enter_OK;
RTE_OK   := LightData.GateLocked AND LightData.Req_To_Enter_OK;
Gates_OK := LightData.AllGatesReset AND LightData.GateLocked AND NOT LightData.MaintMode;
MaintModeActive := LightData.MaintMode AND (LightData.GateUnlocked OR RTE_OK); 

White    := MaintModeActive;
Red      := GateOpen;
Green    := Gates_OK;
Blue     :=(RTE_OK AND NOT LightData.MaintMode) OR RTE_Req;
Flash    := RTE_Req AND NOT RTE_OK;

//Mapping to Outputs
//IF NOT  (Green,Red,Yellow,Blue,Orange,Purple,White) THEN
//    Mapped_SmartLight[0,1,2] := FALSE  ;
//END_IF

IF Green THEN
    Mapped_SmartLight[0] :=TRUE;
    Mapped_SmartLight[1,2] :=FALSE;
END_IF

IF Red THEN
    Mapped_SmartLight[1] :=TRUE;
    Mapped_SmartLight[0,2] :=FALSE;
END_IF

IF Yellow THEN
    Mapped_SmartLight[0,1] :=TRUE;
    Mapped_SmartLight[2] :=FALSE;
END_IF

IF Blue THEN
    Mapped_SmartLight[2] :=TRUE;
    Mapped_SmartLight[0,1] :=FALSE;
END_IF

IF Orange THEN
    Mapped_SmartLight[0,2] :=TRUE;
    Mapped_SmartLight[1] :=FALSE;
END_IF

IF Purple THEN
    Mapped_SmartLight[0,1] :=TRUE;
    Mapped_SmartLight[2] :=FALSE;
END_IF

IF White THEN
    Mapped_SmartLight[0,1,2] :=TRUE;
END_IF

IF Flash THEN
    Mapped_SmartLight[3] :=TRUE;
END_IF

*)

END_FUNCTION_BLOCK

// ---- POUs/Cell/Faulthistory_FB.TcPOU
FUNCTION_BLOCK Faulthistory_FB EXTENDS FB_Cell
VAR_INPUT
END_VAR
VAR_OUTPUT
END_VAR
VAR
END_VAR

END_FUNCTION_BLOCK

// ---- POUs/Cell/FB_Cell.TcPOU
FUNCTION_BLOCK FB_Cell
VAR
	fbMainAirDump			  : FB_ActuatorSimple;
    stGate1                   : ST_Gates;
    stGate2                   : ST_Gates;
    fbOp_Smartlight           : FB_BNI007T;
    fbGate1_SmartLight        : FB_BNI007T;
	fbGate2_SmartLight        : FB_BNI007T;
    fbStation_TAP             : FB_TAP;
    stCell	                  : ST_Cell;       //Cell Level 
    stStation                 : ST_Station;   //Station Level
END_VAR

M_Utilities();
M_Power();
M_Modes();
M_Status();
M_AllGateEntry();
M_GateBox();
M_IndicatorLights();

METHOD PUBLIC M_AllGateEntry
VAR_INST
    Request_Timeout_TMR       : TON; //Request to Enter Timeout Timer
    Request_Timeout_TmrDN     : BOOL; //Request to enter timer is Done
END_VAR
//Cell Gate Entry - Control Section

//Request to Enter
IF GVL.stCell.Gates.DoorReqtoEnterInput[1] OR GVL.stCell.Gates.DoorReqtoEnterInput[2] THEN
    GVL.stCell.Gates.Request_To_Enter := TRUE;
        ELSIF   GVL.stCell.Gates.DoorPowerOn[1] OR GVL.stCell.Gates.DoorPowerOn[2] THEN
    GVL.stCell.Gates.Request_To_Enter := FALSE; 
END_IF

//Ok to Enter - All stations and Testing Unit
GVL.stCell.Gates.OK_To_Enter := GVL.stCell.Gates.Request_To_Enter AND GVL.zz_Deep.1;       //Need to add in standard code (After getting each station information)

//Gate entry Granted - Unlock all Gates
Request_Timeout_TMR (IN := GVL.stCell.Gates.Request_To_Enter AND NOT GVL.stCell.Gates.EntryGranted, PT := T#45S, Q => Request_Timeout_TmrDN ); 

GVL.stCell.Gates.EntryGranted := GVL.stCell.Gates.Request_To_Enter AND 
                                        (GVL.stCell.Gates.OK_To_Enter OR 
                                                GVL.stCell.Gates.EntryGranted OR 
                                                            Request_Timeout_TmrDN) ;
END_METHOD

METHOD M_DisplayFaults : BOOL
VAR_INPUT
END_VAR
END_METHOD

METHOD M_DisplayMessages : BOOL
VAR_INPUT
END_VAR
END_METHOD

METHOD M_Faulthistory : BOOL
VAR_INPUT
    COP_Dynamic_String_120_0: COP_Dynamic_String_120;
    COP_Dynamic_String_120_1: COP_Dynamic_String_120;
	COP_Dynamic_String_120_2: COP_Dynamic_String_120;
	COP_Dynamic_String_120_3: COP_Dynamic_String_120;
	COP_Dynamic_String_120_4: COP_Dynamic_String_120;
	COP_Dynamic_String_120_5: COP_Dynamic_String_120;
    COP_Dynamic_String_15_0: COP_Dynamic_String_15;
    COP_Dynamic_String_15_1: COP_Dynamic_String_15;
	COP_Dynamic_String_15_2: COP_Dynamic_String_15;
	COP_Dynamic_String_15_3: COP_Dynamic_String_15;
	COP_Dynamic_String_15_4: COP_Dynamic_String_15;
	COP_Dynamic_String_15_5: COP_Dynamic_String_15;
	FLT_CNT: BYTE := 0;
    Len: BYTE;
    DStart_Pos: DINT;
    Pointr: BYTE;
	History_Temp: ARRAY [0..49] OF STRING(120);
	History_Time_Temp: Array [0..49] of string(15);
	History_Buffer_Temp: Array [0..49] of string(120);
	History_Time_Buffer_Temp: Array [0..49] of string(15);
	FLL1_String_120_0: FLL1_String_120;
	FLL1_String_120_1: FLL1_String_120;
	FLL1_String_15_0: FLL1_String_15;
	FLL1_String_15_1: FLL1_String_15;
END_VAR
IF FLT_CNT>49 THEN
	FLT_CNT:=49;
END_IF

//Initialize Lengths
Len:=49-FLT_CNT;
DStart_Pos:=FLT_CNT;
(*
IF Cell_HMI1.Req.FaultReset=TRUE AND FLT_CNT>0 THEN
	
	//Index Old Fault
	COP_Dynamic_String_120_0(Source:=Cell_HMI1.Fault.History, Dest:=History_Temp, SStart:=0, DStart:=0, Length:= Len);
	COP_Dynamic_String_120_1(Source:=History_Temp, Dest:=Cell_HMI1.Fault.History, SStart:=0, DStart:=DStart_Pos, Length:= Len);
	
	//Index Old Time
	COP_Dynamic_String_15_0(Source:=Cell_HMI1.Fault.History_Time, Dest:=History_Time_Temp, SStart:=0, DStart:=0, Length:= Len);
	COP_Dynamic_String_15_1(Source:=History_Time_Temp, Dest:=Cell_HMI1.Fault.History_Time, SStart:=0, DStart:=DStart_Pos, Length:= Len);
	
	// Copy New Faults
	COP_Dynamic_String_120_2(Source:=Cell_HMI1.Fault.History_Buffer, Dest:=Cell_HMI1.Fault.History, SStart:=0, DStart:=0, Length:= FLT_CNT-1);
	
	// Copy New Time
	COP_Dynamic_String_15_2(Source:=Cell_HMI1.Fault.History_Time_Buffer, Dest:=Cell_HMI1.Fault.History_Time, SStart:=0, DStart:=0, Length:= FLT_CNT-1);
	
	//Clear All Data
	FLL1_String_120_0(Dest:=Cell_HMI1.Fault.History_Buffer , Source:= '', Start:= 0, Length:=49 );
	FLL1_String_120_1(Dest:=History_Buffer_Temp , Source:= '', Start:= 0, Length:=49 );
	FLL1_String_15_0(Dest:=Cell_HMI1.Fault.History_Time_Buffer , Source:= '', Start:= 0, Length:=49 );
	FLL1_String_15_1(Dest:=History_Time_Buffer_Temp , Source:= '', Start:= 0, Length:=49 );
	
	//Reset Fault Count
	FLT_CNT:=0;
	
END_IF

IF Cell_HMI1.Fault.Display<>'' THEN
IF FLT_CNT<=49 THEN			
				Pointr:=0;
				WHILE Pointr<=49 DO
					IF Cell_HMI1.Fault.History_Buffer[Pointr]=Cell_HMI1.Fault.Display THEN
					   Cell_HMI1.Fault.History_Time_Buffer[Pointr]:=Cell_HMI1.Fault.Current_Time;
					   JMP END;
					END_IF
					Pointr:=Pointr+1;
				END_WHILE
				
     		    //Index Fault Buffer
                COP_Dynamic_String_120_3(Source:=Cell_HMI1.Fault.History_Buffer, Dest:=History_Buffer_Temp, SStart:=0, DStart:=1, Length:= 48);
 				COP_Dynamic_String_120_4(Source:=History_Buffer_Temp, Dest:=Cell_HMI1.Fault.History_Buffer, SStart:=1, DStart:=1, Length:= 48);
				
				//Index Time Buffer
				COP_Dynamic_String_15_3(Source:=Cell_HMI1.Fault.History_Time_Buffer, Dest:=History_Time_Buffer_Temp, SStart:=0, DStart:=1, Length:= 48);
				COP_Dynamic_String_15_4(Source:=History_Time_Buffer_Temp, Dest:=Cell_HMI1.Fault.History_Time_Buffer, SStart:=1, DStart:=1, Length:= 48);
				
				//Copy Fault and Time To the First Buffer Position				
				Cell_HMI1.Fault.History_Buffer[0]:=Cell_HMI1.Fault.Display;
				Cell_HMI1.Fault.History_Time_Buffer[0]:=Cell_HMI1.Fault.Current_Time;
				FLT_CNT:=FLT_CNT+1;
END_IF						
END_IF
*)
//End:
END_METHOD

METHOD PRIVATE M_GateBox
VAR
END_VAR
//GateBox-1 Lock Solenoid
(*
IF GVL.Cell.Gates.DoorReqtoEnterInput[1] AND GVL.Cell.Gates.Request_To_Enter THEN
    GVL.Cell.Gates.DoorUnlockRequest[1] := TRUE;
ELSIF GVL.Cell.Gates.DoorPowerOn[1] AND  GVL.zz_Deep.0 AND GVL.zz_Deep.0 THEN
    GVL.Cell.Gates.DoorUnlockRequest[1] := FALSE;
END_IF

GVL.Cell.Gates.DoorOktoUnlock[1] := (GVL.Cell.Gates.EntryGranted OR 
                                          GVL.Cell.Gates.DoorOktoUnlock[1] OR 
                                          GVL.zz_Deep.0)  AND 
                                          GVL.Cell.Gates.DoorUnlockRequest[1];
                                         
//GateBox-1 - Smart light Mapping
//White Light
GVL.Cell.Gates.ReqtoEnterInput_LT[1] :=  GVL.Cell.Gates.DoorUnlockRequest[1] AND 
                                            GVL.Cell.Gates.Request_To_Enter AND 
                                            GVL.Cell.Gates.OK_To_Enter AND 
                                            GVL.Cell.Gates.EntryGranted AND 
                                            (NOT Gate1.Maintenance_Mode OR (Gate1.Maintenance_Mode AND Gate1.Teach_Mode_OK));  

//Green Liight

GVL.Cell.Gates.FaultResetInput_LT[1] :=  (Gate1.Reset OR (Gate1.closed AND NOT Gate1.Reset AND Gate1.Maintenance_Mode) AND 
                                            (NOT Gate1.Maintenance_Mode OR (Gate1.Maintenance_Mode AND Gate1.Teach_Mode_OK)))  OR
                                            (Gate1.Maintenance_Mode AND NOT Gate1.Teach_Mode_OK);                                         
                                            
//Red Light
GVL.Cell.Gates.FaultResetInput_LT[1] :=  (GVL.Cell.Status.All_Faults AND 
                                            ( NOT Gate1.Maintenance_Mode OR (Gate1.Maintenance_Mode AND Gate1.Teach_Mode_OK))) OR
                                            Gate1.DoorFaultResetInput[1]   OR
                                            (Gate1.Maintenance_Mode AND NOT Gate1.Teach_Mode_OK);
                                            

                                            
                                            
                                            
                                            
//GateBox-2 Lock Solenoid
IF GVL.Cell.Gates.DoorReqtoEnterInput[2] AND GVL.Cell.Gates.Request_To_Enter THEN
    GVL.Cell.Gates.DoorUnlockRequest[2] := TRUE;
ELSIF GVL.Cell.Gates.DoorPowerOn[1] AND  GVL.zz_Deep.0 AND GVL.zz_Deep.0 THEN
    GVL.Cell.Gates.DoorUnlockRequest[2] := FALSE;
END_IF

GVL.Cell.Gates.DoorOktoUnlock[2] := (GVL.Cell.Gates.EntryGranted OR 
                                          GVL.Cell.Gates.DoorOktoUnlock[2] OR 
                                          GVL.zz_Deep.0)  AND 
                                          GVL.Cell.Gates.DoorUnlockRequest[2];

//GateBox-2 - Smart light Mapping
//White Light
GVL.Cell.Gates.ReqtoEnterInput_LT[2] :=  GVL.Cell.Gates.DoorUnlockRequest[2] AND 
                                            GVL.Cell.Gates.Request_To_Enter AND 
                                            GVL.Cell.Gates.OK_To_Enter AND 
                                            GVL.Cell.Gates.EntryGranted AND 
                                            (NOT Gate2.Maintenance_Mode OR (Gate2.Maintenance_Mode AND Gate2.Teach_Mode_OK));  

//Green Liight
GVL.Cell.Gates.FaultResetInput_LT[2] :=  (Gate2.Reset OR (Gate2.closed AND NOT Gate2.Reset AND Gate2.Maintenance_Mode) AND 
                                            (NOT Gate2.Maintenance_Mode OR (Gate2.Maintenance_Mode AND Gate2.Teach_Mode_OK)))  OR
                                            (Gate2.Maintenance_Mode AND NOT Gate2.Teach_Mode_OK);
                                            
                                            
//Red Light
GVL.Cell.Gates.FaultResetInput_LT[2] :=  (GVL.Cell.Status.All_Faults AND 
                                            ( NOT Gate2.Maintenance_Mode OR (Gate2.Maintenance_Mode AND Gate2.Teach_Mode_OK))) OR
                                            Gate2.DoorFaultResetInput   OR
                                            (Gate2.Maintenance_Mode AND NOT Gate2.Teach_Mode_OK) ;                                          
                                            *)
END_METHOD

METHOD M_IndicatorLights
VAR_INPUT
END_VAR
END_METHOD

METHOD M_MessageHistroy : BOOL
VAR_INPUT
END_VAR
END_METHOD

METHOD PRIVATE M_Modes
VAR_INST
    PowerdownTmr    : TON;  //Auto Power off After 1 Hour of sitting idle
END_VAR
// Cell Modes - Control Section

//Auto-Manual Mode Sleector Switch
GVL.stCell.stMode.AutoSelect_Toggle.Toggle  := GVL.stCell.PV_PB.AutoManual_SS;
                                          
IF (GVL.stCell.stMode.AutoSelect_Toggle.Toggle AND NOT GVL.stCell.stMode.AutoSelect_Toggle.On ) OR 
     (NOT GVL.stCell.stMode.AutoSelect_Toggle.Toggle AND GVL.stCell.stMode.AutoSelect_Toggle.On ) THEN
          GVL.stCell.stMode.AutoSelect_Toggle.On :=TRUE;
          ELSE  
          GVL.stCell.stMode.Manual :=TRUE;
		  END_IF;   
                                                                                                                                  
GVL.stCell.stMode.Autoinitiate   :=GVL.stCell.PV_PB.AutoMode_PB;

//GVL.Cell.Mode.Manual := NOT GVL.Cell.Mode.AutoSelect_Toggle.On; 
//GVL.Cell.Mode.AutoSelect_Toggle.On := (GVL.Cell.Mode.AutoSelect_Toggle.Toggle AND NOT GVL.Cell.Mode.AutoSelect_Toggle.On ) OR (NOT GVL.Cell.Mode.AutoSelect_Toggle.Toggle AND GVL.Cell.Mode.AutoSelect_Toggle.On );
                                           
// Cell Automatic Run Mode
GVL.zz_Deep.1 := TRUE;                      //Need to add in standard code
 
//Auto Power off
GVL.zz_Deep.1 := TRUE;                      //Need to add in standard code
END_METHOD

METHOD PUBLIC M_Power
VAR_INST
	CtrlPwrOnTmr : TON;      //Control Power ON Timer
END_VAR
//Cell Specific General Safeties
(*
GVL.Cell.Power.Gen_Safety := GVL.Cell.Power.PowerOn AND 
								GVL.Cell.Power.GatesClosed AND 
								GVL.Cell.Utility.MainAirOn AND 
								GVL.Cell.Status.AllComms_OK;


//Control Power ON
CtrlPwrOnTmr (IN := GVL.Cell.Power.EStops , PT := T#125MS, Q => GVL.Cell.Power.PowerOn); 

//No E-Stops Pressed
GVL.zz_Deep.0 := TRUE;                   //Need to add once get safety code

//AllZone Gates are closed
GVL.zz_Deep.0 := TRUE;                  //Need to add once get safety code

  


*)
END_METHOD

METHOD PUBLIC M_ResetFault
VAR_INPUT
END_VAR
fbStation_TAP.M_ResetFault();
END_METHOD

METHOD PRIVATE M_Status
VAR_INST
    FaultResetTmr : TON;
    CommsOKTmr    : TON; // All Communication Modules OK Delay Off Timer
END_VAR
// Cell Status - Control Selection
FaultResetTmr (IN := GVL.stCell.PV_PB.FaultReset_PB OR GVL.stCell.Gates.DoorFaultResetInput[1] OR GVL.stCell.Gates.DoorFaultResetInput[2] , PT := T#0.1S, Q => GVL.stCell.Status.Fault_Reset);                                                                                                                       

// All Cell Level Comms OK
CommsOKTmr (IN := GVL.stCell.Status.ENetComms_OK, PT := T#1S, Q => GVL.stCell.Status.AllComms_OK ); 

//All Zone Level - EtherCAT Modules OK
GVL.zz_Deep.1 := TRUE;                      //Need to add in standard code


//Station Signals used in Zone Level
//All Station -Fault Present

GVL.stCell.Status.All_Faults := GVL.stCell.Status.Faulted OR GVL.stStation.Status.Faulted OR GVL.zz_Deep.1; 

//All Station - Messages Present

GVL.stCell.Status.Message    := GVL.stCell.Status.Message OR GVL.stStation.Status.Message OR GVL.zz_Deep.1;
END_METHOD

METHOD PRIVATE M_TAP
VAR_INPUT
END_VAR
fbStation_TAP(stCell := stCell);
END_METHOD

METHOD PRIVATE M_Utilities
VAR_INST
	AirOnTmr	: TON;
	AirOffTmr	: TON;	
END_VAR
// Main Air Dump
IF GVL.stCell.stPower.PowerOn THEN
	fbMainAirDump.M_Advance();
ELSE
	fbMainAirDump.M_Retract();
END_IF

// Air Pressure OK
AirOffTmr (IN := GVL.stCell.stUtility.MainAirPSI < 70, PT := T#2S);
AirOnTmr (IN := GVL.stCell.stUtility.MainAirPSI >= 90 AND NOT AirOffTmr.Q, PT := T#1.5S, Q => GVL.stCell.stUtility.MainAirOn);
END_METHOD

END_FUNCTION_BLOCK

// ---- POUs/Station/TAP/FB_TAP.TcPOU
FUNCTION_BLOCK FB_TAP
VAR_INPUT    
    stCell                          : REFERENCE TO ST_Cell;
END_VAR
VAR
	TAP_LevelSensor AT%I*	        : DINT;                     //Level Sensor
    TAP_TempSensor AT%I*            : DINT;                     //Temp in Celsius
	TE_TapPressureSensor_PT1 AT%I*    : INT;                      //Pressure Sensor in PSI 
    TE_TapPressureSensor_PT2 AT%I*    : INT;                      //   
    fbtapmotor                      : FB_Motor;                 //HPU Motor
	SolenoidFluidValve_SVD1A        : FB_ActuatorSimple;
    SolenoidFluidValve_SVD1B        : FB_ActuatorSimple;
    SolenoidFluidValve_SP2          : FB_ActuatorSimple;
    stTAPStation                    : ST_Station;
    stTAPSta_HMI                    : ST_TAP_PB;
    
END_VAR

M_Motor();

METHOD M_Faults : BOOL
VAR_INPUT
END_VAR
END_METHOD

METHOD PRIVATE M_LevelSensor : BOOL
VAR_INPUT
END_VAR
END_METHOD

METHOD M_Monitor : BOOL
VAR_INPUT
END_VAR
END_METHOD

METHOD PRIVATE M_Motor
VAR_INPUT
END_VAR
fbtapmotor.SafetyOk := stCell.Safety.SafetyOk;
fbtapmotor();

IF HMI.MotorStartPB AND ManualOK THEN
fbtapmotor.M_Start();
ELSIF HMI.MotorStopPB THEN
    fbtapmotor.M_Stop();
END_IF
END_METHOD

METHOD PUBLIC M_ResetFault
VAR_INPUT
END_VAR
fbtapmotor.M_ResetFault();
END_METHOD

METHOD PRIVATE M_Sequence
VAR_INPUT
	AutoInitiate 	    : BOOL;
	AutoFirstStep	    : DINT;
END_VAR                 
VAR_INST                
	fbSequenceStep		       : FB_SequenceStep;
	FirstEntry		           : BOOL := TRUE;
	(*CaseEntry		           : ARRAY [1..20] OF BOOL := [20(TRUE)];*)
	PressureAtEntryP1 AT%I*    : INT;         //P1 Pressure in PSI for UUT
    PressureAtExitP2  AT%I*    : INT;        // P2 Pressure in PSI for UUT
    Maxtemp                    : INT :=110;   //Max temp setup value
    InitialPressurePT1         : INT :=30;    //Initial Pressure PT1      
    ExpectedPressureP1         : INT;        // P1 Expected pressure UP1 in PSI_COnstant Value
    ExpectedPressureP2         : INT;        // P2 Expected pressure UP2 in PSI_COnstant Value
    PressuredropPF             : INT;        // Pressure Drop thorugh Filter_Contant Value
    PressureCheckStatus        : INT;        // Pressure Check Value
    SensorCheckStatus          : INT;        // Sensor Check Value and status 
    CheckValveStatus           : INT;        // Valve Check Value and Status 
    FailedintitialPressure     : INT;        // Initial Pressure check failed  
    Tolerance                  : INT;        
	FailReasonStr	           : STRING;     // Reason for Test Fail 
    PassReasonStr              : STRING;     // Preason for Test Pass 
    FailPressureStr            : STRING;     // Pressure Fail Test Reason 
    FillingupComplete          : STRING;     //Process Complete  
    TEtapstarttimer            : TON;        // Tap Test Start timer   
    TEMotorTimer               : TON;        // Tap TE-HPU motor start timer
    TEMOtorruntimer            : TON;        // Tap TE-HPU motor running timer
    TEmotorostoptimer          : TON;        // Tap TE-HPU motor stop timer
    UUTmotorONtimer            : TON;        // Tap UUT-motor timer on 
    UUTmotorOFFtimer           : TON;        // Tap UUT-motor timer off 
    LeakDecayTimer             : TON;        // Leak Delay Timer
    DrainONTimer               : TON;        // System Drain Timer
END_VAR                        
VAR                            
    Branch                     : ARRAY [1..16] OF ST_StepBranch;
END_VAR
IF FirstEntry THEN
	fbSequenceStep.CurrentStep := AutoFirstStep;
END_IF

IF AutoInitiate THEN
FirstEntry := FALSE;
CASE fbSequenceStep.CurrentStep OF
	E_TapAutoSequenceSteps.STARTING_CONDITIONS:
		IF fbSequenceStep.Entry THEN
            SolenoidFluidValve_SP2.M_Retract();
            SolenoidFluidValve_SVD1A.M_Retract();
            SolenoidFluidValve_SVD1B.M_Advance();            
		END_IF
        
        // Execute During
        TEtapstarttimer(IN := FALSE);
        TEtapstarttimer(IN := TRUE, PT := T#500MS);
                
        // Branch #1
        Branch[1].NextStep     := E_TapAutoSequenceSteps.TE_RUN_MOTOR;
        Branch[1].Condition[1] := stTAPStation.Status.AllParts;
        Branch[1].Condition[2] := (TAP_TempSensor < Maxtemp) AND (TE_TapPressureSensor_PT1<InitialPressurePT1);
        Branch[1].Condition[3] := SolenoidFluidValve_SP2.stStatus.RetractedFeedback;
        Branch[1].Condition[4] := SolenoidFluidValve_SVD1A.stStatus.RetractedFeedback;
        Branch[1].Condition[5] := SolenoidFluidValve_SVD1B.stStatus.AdvancedFeedback;
        Branch[1].Condition[6] := TEtapstarttimer.Q AND NOT TEMOtorruntimer.Q;
        Branch[1].Condition[7] := GVL.zz_Deep.0; //Need to add condition for UUT Unit
        
        fbSequenceStep(Branch := Branch);

	E_TapAutoSequenceSteps.TE_RUN_MOTOR:
		// Action
		IF fbSequenceStep.Entry THEN
		fbtapmotor.M_Start();
		END_IF
        
        TEMOtorruntimer(IN := FALSE);
        TEMOtorruntimer(IN := TRUE, PT := T#5S);
                
        // Branch #1
        Branch[1].NextStep     := E_TapAutoSequenceSteps.START_UUT_MOTOR;
        Branch[1].Condition[1] := stTAPStation.Status.Auto AND stCell.Status.All_in_Auto;
        Branch[1].Condition[2] := TEMOtorruntimer.Q;
        Branch[1].condition[3] := fbtapmotor.stmotorinputs.Running; //Need to add contion for input that TE motor is running
        Branch[1].Condition[4] := //Need to add extra conditon to check UUt Motor 
               
        fbSequenceStep(Branch := Branch);
        
	E_TapAutoSequenceSteps.START_UUT_MOTOR:	
        //Action
        IF fbSequenceStep.Entry THEN
         ///Condition for next step: UUT MOTOR RAMP-UP TO SPEED= "UMLS" 
		END_IF
        
        // Branch #1
        Branch[1].NextStep     := E_TapAutoSequenceSteps.UUT_MOTOR_DELAY;
        Branch[1].Condition[1] := //Need to add extra condition TO EXECUTE UUT MOTOR DELAY            
 
        fbSequenceStep(Branch := Branch);
        
	E_TapAutoSequenceSteps.UUT_MOTOR_DELAY:
		// Action
		IF fbSequenceStep.Entry THEN
		//Condition for next step: UUT Motor Ramp-up to speed; "UMD1"
        END_IF
        
        UUTmotorONtimer(IN := FALSE);
        UUTmotorONtimer(IN := TRUE, PT := T#5S);
        
         // Branch #1
        Branch[1].NextStep     := E_TapAutoSequenceSteps.INITIAL_PRESSURE_TEST;
        Branch[1].Condition[1] := UUTmotorONtimer.Q;
        Branch[1].Condition[2] := //condition needs to add: Motor speed for filling needs to 100RPm and time delay needs to 5_10 seconds
                          
        fbSequenceStep(Branch := Branch);
         
    E_TapAutoSequenceSteps.INITIAL_PRESSURE_TEST:
        // Action         
        LeakDecayTimer(IN := PressureAtEntryP1 = ExpectedPressureP1 + Tolerance OR ExpectedPressureP1 - Tolerance , PT := T#5S);
        IF  LeakDecayTimer.Q THEN
        IF ExpectedPressureP1 < PressureAtEntryP1 - Tolerance OR ExpectedPressureP1 > PressureAtEntryP1 + Tolerance THEN
		PressureCheckStatus := E_PressureStatus.FillingupTestFail;
		FailReasonStr := TO_STRING(E_PressureStatus.FillingupTestFail);
       	ELSE
		PressureCheckStatus := E_PressureStatus.FillingupTestPass;
        PassReasonStr := TO_STRING(E_PressureStatus.FillingupTestPass); 
       	END_IF
	    END_IF    
              
         // Branch #1
        Branch[1].NextStep     := E_TapAutoSequenceSteps.COMPLETE ;
        Branch[1].Condition[1] := PressureCheckStatus := 10;
 
         // Branch #2 (Move to Next test)
        Branch[2].NextStep     := E_TapAutoSequenceSteps.TE_STOP_MOTOR ;
        Branch[2].Condition[1] := PressureCheckStatus := 20;
                      
        fbSequenceStep(Branch := Branch);
        
	E_TapAutoSequenceSteps.TE_STOP_MOTOR:
		// Action
		IF fbSequenceStep.Entry THEN
		   fbtapmotor.M_Stop();
		END_IF
        
        TEmotorostoptimer( IN:= FALSE );
        TEmotorostoptimer( IN:= TRUE ,PT := T#5S);
        
         // Branch #1
        Branch[1].NextStep     := E_TapAutoSequenceSteps.STOP_UUT_MOTOR;
        Branch[1].Condition[1] := NOT fbtapmotor.st_motorinputs.Running;
        Branch[1].Condition[2] := TEmotorostoptimer.Q;       
       
        fbSequenceStep(Branch := Branch); 
               
    E_TapAutoSequenceSteps.STOP_UUT_MOTOR:
        //Action
        IF (*add action to stoppped UUt motor*)     THEN     //Condition for next Setp: Stop UUT Motor
        END_IF
        
        UUTmotorOFFtimer ( IN:= FALSE );
        UUTmotorOFFtimer (IN:= TRUE , PT := T#5S);

         // Branch #1
        Branch[1].NextStep     := E_TapAutoSequenceSteps.END_FILLING_PHASE ;
        Branch[1].Condition[1] := (PressureCheckStatus := 10) AND NOT (PressureCheckStatus := 20);
        Branch[1].Condition[2] := UUTmotorOFFtimer.Q;
                

        fbSequenceStep(Branch := Branch); 
    
    E_TapAutoSequenceSteps.END_FILLING_PHASE:
        //Action
        IF fbSequenceStep.Entry THEN
        IF NOT fbtapmotor.stmotorinputs.Running AND (*CONDITION FOR UUT TO STOPPED VERIFED*) THEN          
            SolenoidFluidValve_SP2.M_Advance();
            SolenoidFluidValve_SVD1A.M_Retract();
            SolenoidFluidValve_SVD1B.M_Advance();
            FillingupComplete := TO_STRING (E_TapAutoSequenceSteps.END_FILLING_PHASE); 
		END_IF
        END_IF
        
        // Branch #1
        Branch[1].NextStep     := E_TapAutoSequenceSteps.START_STATIC_PRESSURE_TEST;
        Branch[1].Condition[1] := PressureCheckStatus := 20;
        Branch[1].Condition[2] := TAP_TempSensor < Maxtemp AND TE_TapPressureSensor_PT1 > InitialPressurePT1;
        Branch[1].Condition[3] := SolenoidFluidValve_SP2.stStatus.AdvancedFeedback;
        Branch[1].Condition[4] := SolenoidFluidValve_SVD1A.stStatus.RetractedFeedback;
        Branch[1].Condition[5] := SolenoidFluidValve_SVD1B.stStatus.AdvancedFeedback;
        Branch[1].Condition[6] := NOT fbtapmotor.stmotorinputs.Running;

        fbSequenceStep(Branch := Branch); 

    E_TapAutoSequenceSteps.START_STATIC_PRESSURE_TEST:
		// Action
		IF fbSequenceStep.Entry THEN
		fbtapmotor.M_Start();
		END_IF        
        
        TEMOtorruntimer(IN := FALSE);
        TEMOtorruntimer(IN := TRUE, PT := T#5S);
        
      
        // Branch #1
        Branch[1].NextStep     := E_TapAutoSequenceSteps.OUTLET_PRESSURE_TEST;
        Branch[1].Condition[1] := TEMOtorruntimer.Q;
        Branch[1].condition[2] := fbtapmotor.stmotorinputs.Running; //Need to add contion for input that TE motor is running
        Branch[1].Condition[3] := TE_TapPressureSensor_PT2 = ExpectedPressureP2 + Tolerance OR ExpectedPressureP2 - Tolerance;
 
       fbSequenceStep(Branch := Branch); 

    E_TapAutoSequenceSteps.OUTLET_PRESSURE_TEST:
        //Action
        IF  fbSequenceStep.Entry THEN
        IF TE_TapPressureSensor_PT1 = (ExpectedPressureP2 + Tolerance) OR (ExpectedPressureP2 - Tolerance) THEN
            fbtapmotor.M_Stop();            
        END_IF
        END_IF    
        
        TEmotorostoptimer(IN :=FALSE); 
        TEmotorostoptimer(IN:= TRUE ,PT := T#2S);
        
        IF TEmotorostoptimer.Q AND (PressureAtEntryP1 = (ExpectedPressureP2 + Tolerance) OR (ExpectedPressureP2 - Tolerance)) THEN
            PressureCheckStatus := E_PressureStatus.PressuretestOk;
		    PassReasonStr := TO_STRING(E_PressureStatus.PressuretestOk);
        ELSIF PressureAtExitP2 <> ExpectedPressureP2 THEN
                PressureCheckStatus := E_PressureStatus.InletLeakDetect;
                FailReasonStr := CONCAT(CONCAT(TO_STRING(E_PressureStatus.PressuretestOk), ' AND '), TO_STRING(E_PressureStatus.InletLeakDetect));
        ELSIF PressureCheckStatus = E_PressureStatus.OilLeakDetect;
                FailPressureStr := TO_STRING(E_PressureStatus.OilLeakDetect);
			END_IF
        END_IF  
        
        // Branch #1
        Branch[1].NextStep     := E_TapAutoSequenceSteps.COMPLETE;
        Branch[1].Condition[1] := (PressureCheckStatus = E_PressureStatus.InletLeakDetect) OR (PressureCheckStatus = E_PressureStatus.OilLeakDetect);        

        // Branch #2
        Branch[2].NextStep     := E_TapAutoSequenceSteps.END_STAITC_PRESSURE_TEST;
        Branch[2].Condition[1] := PressureCheckStatus = 30 ;
        Branch[2].Condition[2] := TEmotorostoptimer.Q;

        fbSequenceStep(Branch := Branch); 

    E_TapAutoSequenceSteps.END_STAITC_PRESSURE_TEST:
        //Action     
        IF fbSequenceStep.Entry THEN
             SolenoidFluidValve_SP2.M_Advance();
                SolenoidFluidValve_SVD1A.M_Retract();
                   SolenoidFluidValve_SVD1B.M_Retract();       
        END_IF     
     
        // Branch #1
        Branch[1].NextStep     := E_TapAutoSequenceSteps.START_FUNCTIONAL_TEST;
        Branch[1].Condition[1] := TAP_TempSensor < Maxtemp ;
        Branch[1].Condition[2] := SolenoidFluidValve_SP2.stStatus.AdvancedFeedback;
        Branch[1].Condition[3] := SolenoidFluidValve_SVD1A.stStatus.RetractedFeedback;
        Branch[1].Condition[4] := SolenoidFluidValve_SVD1B.stStatus.RetractedFeedback;
        Branch[1].Condition[5] := NOT fbtapmotor.stmotorinputs.Running;
  
        fbSequenceStep(Branch := Branch); 
          
     E_TapAutoSequenceSteps.START_FUNCTIONAL_TEST: 
        //Actiion
        IF fbSequenceStep.Entry THEN
         ///Condition for next step: UUT MOTOR tURN ON AND RAMP-UP TO SPEED= "UMD3" 
 		END_IF

       UUTmotorONtimer(IN := FALSE); 
       UUTmotorONtimer(IN := TRUE, PT := T#5S);

       
         // Branch #1
        Branch[1].NextStep     := E_TapAutoSequenceSteps.UUT_SENSOR_CHECK;
        Branch[1].Condition[2] := UUTmotorONtimer.Q;
        Branch[1].Condition[3] := //condition needs to add: mONITOR Motor speed for filling needs to 100RPm and time delay needs to 5_10 seconds
        
        fbSequenceStep(Branch := Branch); 
       
      E_TapAutoSequenceSteps.UUT_SENSOR_CHECK:
       //Action
       IF fbSequenceStep.Entry THEN
           IF 
               (PressureAtExitP2 < TE_TapPressureSensor_PT1 + Tolerance) OR (PressureAtExitP2 > TE_TapPressureSensor_PT1 - Tolerance) THEN 
               SensorCheckStatus := E_SenorStatus.P2UUTSensorOK;
               PassReasonStr     := TO_STRING(E_SenorStatus.P2UUTSensorOK);
            ELSE
                SensorCheckStatus := E_SenorStatus.P2UUTSensorFail;
                FailReasonStr     := TO_STRING(E_SenorStatus.P2UUTSensorFail);
           END_IF
           
            IF 
               (PressureAtExitP2 = PressureAtEntryP1 - PressuredropPF) THEN
               SensorCheckStatus := E_SenorStatus.P1UUTSensorOK ;
               PassReasonStr     := CONCAT(CONCAT(TO_STRING(E_SenorStatus.P1UUTSensorOK), ' AND '), TO_STRING(E_SenorStatus.Filterisdetected));   
		   END_IF
           
           IF (PressureAtExitP2 < PressureAtEntryP1 + Tolerance) OR (PressureAtExitP2 > PressureAtEntryP1 - Tolerance) THEN
               SensorCheckStatus := E_SenorStatus.Filterismissing;
               FailReasonStr     := TO_STRING(E_SenorStatus.Filterismissing);       
           ELSE
               SensorCheckStatus := E_SenorStatus.P1UUTSensorFail;
               FailReasonStr     := TO_STRING(E_SenorStatus.P1UUTSensorFail);
           END_IF
		   END_IF
	   
          
         // Branch #1
        Branch[1].NextStep     := E_TapAutoSequenceSteps.COMPLETE ;
        Branch[1].Condition[1] := (SensorCheckStatus := 10) OR (SensorCheckStatus := 50) OR (SensorCheckStatus := 20);

          // Branch #1
        Branch[2].NextStep     := E_TapAutoSequenceSteps.END_FUNCTIONAL_TEST;
        Branch[2].Condition[1] := (SensorCheckStatus := 30) OR (SensorCheckStatus :=60); //Verify and needs to add one more value during P1 IS oKAY         
        
        fbSequenceStep(Branch := Branch); 
       
      E_TapAutoSequenceSteps.END_FUNCTIONAL_TEST:
       //Action
       IF fbSequenceStep.Entry THEN
         SolenoidFluidValve_SP2.M_Advance();
            SolenoidFluidValve_SVD1A.M_Advance();
                SolenoidFluidValve_SVD1B.M_Retract();
        END_IF        
        
          // Branch #1
        Branch[1].NextStep     := E_TapAutoSequenceSteps.START_TAP_CHECKVALVE_TEST;
        Branch[1].Condition[1] := SolenoidFluidValve_SP2.stStatus.AdvancedFeedback;
        Branch[1].Condition[2] := SolenoidFluidValve_SVD1A.stStatus.AdvancedFeedback;
        Branch[1].Condition[3] := SolenoidFluidValve_SVD1B.stStatus.RetractedFeedback;
        Branch[1].Condition[4] := NOT fbtapmotor.stmotorinputs.Running;
               
        fbSequenceStep(Branch := Branch); 
       
      E_TapAutoSequenceSteps.START_TAP_CHECKVALVE_TEST:
       //Action
       IF fbSequenceStep.Entry THEN
		fbtapmotor.M_Start();        
	    END_IF
        
        TEMOtorruntimer(IN :=FALSE);
        TEMOtorruntimer(IN := TRUE, PT := T#30S);
                
        // Branch #1
        Branch[1].NextStep     := E_TapAutoSequenceSteps.CHECK_VALVE_TEST;
        Branch[1].Condition[1] := TEMOtorruntimer.Q;
        Branch[1].condition[2] := fbtapmotor.stmotorinputs.Running;
               
        fbSequenceStep(Branch := Branch);            
        
       E_TapAutoSequenceSteps.CHECK_VALVE_TEST:
       //Action
       IF fbSequenceStep.Entry THEN       
          IF ((PressureAtExitP2 < ExpectedPressureP2 + Tolerance) OR (PressureAtExitP2 > ExpectedPressureP2 - Tolerance)) AND PressureAtEntryP1 := 0 THEN
              CheckValveStatus := E_Checkvalvereject.CheckvalveOk;
              PassReasonStr    := TO_STRING(E_Checkvalvereject.CheckvalveOk);
          ELSE
             CheckValveStatus := E_Checkvalvereject.Checkvalvefailure;
             FailReasonStr    := TO_STRING(E_Checkvalvereject.Checkvalvefailure);                
          END_IF  
        END_IF
        
         //Need add logic to store P1, P2 and PT1
                       
         // Branch #1
        Branch[1].NextStep     := E_TapAutoSequenceSteps.END_TAP_CHECKVALVE_TEST;
        Branch[1].condition[1] := fbtapmotor.stmotorinputs.Running; //Need to add contion for input that TE motor is running
        Branch[1].Condition[2] := (CheckValveStatus := 10) OR (CheckValveStatus := 20);
               
        fbSequenceStep(Branch := Branch);            
        
       E_TapAutoSequenceSteps.END_TAP_CHECKVALVE_TEST:
       //Action
       IF fbSequenceStep.Entry THEN
            fbtapmotor.M_Stop();
            TEmotorostoptimer( IN:= fbtapmotor.M_Stop AND NOT fbtapmotor.stmotorinputs.Running ,PT := T#5S);
        END_IF
	        
       IF TEmotorostoptimer.Q THEN
          SolenoidFluidValve_SP2.M_Retract();
          SolenoidFluidValve_SVD1A.M_Retract();
          SolenoidFluidValve_SVD1B.M_Advance();
          //Condition for next step: UUT Motor Ramp-up to speed; "UMD1"
        UUTmotorONtimer(IN := (*NEED TO ADD COMPLETE CONDITION *)AND NOT UUTmotorOFFtimer.Q, PT := T#5S);
       END_IF         		
       
         // Branch #1
        Branch[1].NextStep     := E_TapAutoSequenceSteps.START_DRAINING_TEST;
        Branch[1].Condition[1] := UUTmotorONtimer.Q;
        Branch[1].Condition[2] := NOT fbtapmotor.stmotorinputs.Running; //Need to add contion for input that TE motor is running
        Branch[1].Condition[3] := SolenoidFluidValve_SP2.stStatus.RetractedFeedback;
        Branch[1].Condition[4] := SolenoidFluidValve_SVD1A.stStatus.RetractedFeedback;
        Branch[1].Condition[5] := SolenoidFluidValve_SVD1B.stStatus.AdvancedFeedback;
        
        fbSequenceStep(Branch := Branch);            
        
       E_TapAutoSequenceSteps.START_DRAINING_TEST:
       //Action
       IF fbSequenceStep.Entry THEN                       
           DrainONTimer (IN:= TRUE, PT:= T#5S);
       END_IF
 
        // Branch #1
        Branch[1].NextStep     := E_TapAutoSequenceSteps.COMPLETE;
        Branch[1].Condition[1] := DrainONTimer.Q;
    //  Branch[1].Condition[2] := (PressureCheckStatus := 10) OR (PressureCheckStatus := 50) OR (PressureCheckStatus := 60);
    //  Branch[1].Condition[3] := (E_SenorStatus := 40); 
                        
        fbSequenceStep(Branch := Branch); 
        
       E_TapAutoSequenceSteps.COMPLETE:
       //Action
       IF fbSequenceStep.Entry THEN 
         fbtapmotor.M_Stop()
         (*UUT Motor needs to stop*)
         SolenoidFluidValve_SP2.M_Retract();
            SolenoidFluidValve_SVD1A.M_Retract();
                SolenoidFluidValve_SVD1B.M_Advance();       
       END_IF
END_CASE

END_IF
END_METHOD

METHOD PRIVATE M_TransmissionFluidPressure : BOOL
VAR_INPUT
END_VAR
END_METHOD

METHOD PRIVATE M_TransmissionFluidValve
VAR
END_VAR
END_METHOD

END_FUNCTION_BLOCK

// ---- POUs/SequenceStep_FB/SequenceStep_FB.TcPOU
FUNCTION_BLOCK SequenceStep_FB
VAR_INPUT
    Branch          : ARRAY [1..16] OF ST_StepBranch;
END_VAR
VAR_OUTPUT    
    CurrentStep     : DINT;    
    Entry           : BOOL := TRUE;
END_VAR
VAR
    i : SINT;
    j : SINT;
    Firstscan : BOOL := TRUE;
END_VAR

Entry := FALSE;

IF FirstScan THEN
    Initialize:
    FOR i:= 1 TO 16 DO
        FOR j:= 1 TO 16 DO
            Branch[i].Condition[j] := TRUE;
        END_FOR    
	END_FOR
    Firstscan := FALSE; 
    RETURN;   
END_IF

FOR i:= 1 TO 16 DO
    Branch[i].ConditionMet := TRUE;
    FOR j:= 1 TO 16 DO        
        Branch[i].ConditionMet := Branch[i].Condition[j] AND Branch[i].ConditionMet;
	END_FOR
    IF Branch[i].ConditionMet THEN        
        CurrentStep := Branch[i].NextStep;
        Entry := TRUE;
        JMP Initialize;
	END_IF
    //
END_FOR

END_FUNCTION_BLOCK
